# EPICS autosave request: iocs/PICamIOC/iocBoot/iocPICam/auto_settings.req
file "PICam_settings.req",  P=$(P),  R=cam1:
file "ADBase_settings.req",       P=$(P),  R=cam1:
file "NDPluginBase_settings.req", P=$(P),  R=image1:
file "NDStdArrays_settings.req",  P=$(P),  R=image1:
file "commonPlugin_settings.req", P=$(P)
file "NDFileIMM_settings.req", P=$(P), R=IMM:
